PROGRAM Socket
VAR
	fbFRSocket:fb_socket_FR;
END_VAR

fbFRSocket();

END_PROGRAM

(* stored: Version 1.1.0.1, ProductVersion 3.1.4024.11
   POU Socket: Id {3ea1f794-102b-4ade-8899-710f8bdc81c0}, SpecialFunc None *)
